FUNCTION_BLOCK FB_Safety IMPLEMENTS I_Safety
VAR
	_stSafety : REFERENCE TO ST_SafetyStruct;
END_VAR

METHOD Run : BOOL
VAR_INPUT
END_VAR
END_METHOD

PROPERTY stSafety : REFERENCE TO ST_SafetyStruct
GET
stSafety REF= _stSafety;
END_GET
SET
_stSafety REF= stSafety;
END_SET
END_PROPERTY

END_FUNCTION_BLOCK

(* stored: Version 1.1.0.1, ProductVersion 3.1.4024.11
   POU FB_Safety: Id {951d67ed-7884-467d-be2d-67c25b0a9587}, SpecialFunc None
   Method Run: Id {64e083b8-15a1-49da-b210-79c547f94fed}
   Property stSafety: Id {1d719c29-c6b2-49f9-9c4a-ba307de1077a}
   Get Get: Id {19f5aa76-9bd4-477d-97c9-e2ed42174ee8}
   Set Set: Id {00da6228-5bf2-4ec4-b02d-2a822a9ffc63} *)
